FUNCTION_BLOCK FB_Tote_Subsystem
VAR_INPUT
END_VAR
VAR_OUTPUT
END_VAR
VAR
	status	: MachineStatus := MachineStatus.STOPPED;
	workflow_status	: ToteSubsystemWorkflowStatus := ToteSubsystemWorkflowStatus.UNKNOWN;
	error_status	: OrderToteErrorStatus := OrderToteErrorStatus.UNKNOWN;
	loading_tote	: FB_ToteData;
	buffer_tote		: FB_ToteData;
	working_tote	: FB_ToteData;
	machine_control_cmd	: MachineControlCommand;

	cmd	: OrderToteCommand;
	iLoad	: INT;
	iUnload	: INT;
	ton1	: TON;
	working_tote_status	: ToteStatus;
	p_eTransfer_working	: POINTER TO E_Transfer;

END_VAR


//status					:= GVL.machine_status;
workflow_status			:= GVL.fb_working.workflow_status;
error_status			:= GVL.fb_working.error_status;
working_tote._status	:= GVL.fb_working.tote_status;

p_eTransfer_working	:= ADR(GVL.fb_working.eTransfer);
CASE cmd OF
	OrderToteCommand.DO_NOTHING:
		p_eTransfer_working^	:= E_Transfer.IDLE;
	OrderToteCommand.LOAD:
		p_eTransfer_working^	:= E_Transfer.LOAD;
		IF GVL.fb_working.M_load() THEN
			cmd	:= OrderToteCommand.DO_NOTHING;
		END_IF
	OrderToteCommand.OPEN_BAG:
		workflow_status := ToteSubsystemWorkflowStatus.BAG_OPENING;
		working_tote._status	:= ToteStatus.READY;
		workflow_status := ToteSubsystemWorkflowStatus.IDLE;
		IF GVL.fb_working.M_bag_open() THEN
			cmd	:= OrderToteCommand.DO_NOTHING;
		END_IF
		
	;
	OrderToteCommand.STOP:
		working_tote._status	:= ToteStatus.EMPTY;
		workflow_status := ToteSubsystemWorkflowStatus.IDLE;
		cmd	:= OrderToteCommand.DO_NOTHING;
		;
	OrderToteCommand.SWAP:
		IF M_Unload() THEN
			IF M_Load() THEN
				cmd	:= OrderToteCommand.DO_NOTHING;
			END_IF
		END_IF
	;
	OrderToteCommand.UNLOAD:
		p_eTransfer_working^	:= E_Transfer.UNLOAD;
		IF GVL.fb_working.M_unload() THEN
			cmd	:= OrderToteCommand.DO_NOTHING;
		END_IF
	;	
END_CASE
ton1(PT:=T#1S);

METHOD M_Load : BOOL
VAR_INPUT
END_VAR
M_Load	:=FALSE;
CASE iLoad OF
	0:	
		working_tote._status	:= ToteStatus.EMPTY;
		workflow_status := ToteSubsystemWorkflowStatus.WAITING_FOR_NEW_TOTE;
		ton1.IN	:= FALSE;
		//GVL.iLoad	:= 1;
	1:
		ton1.IN	:= TRUE;
		IF ton1.Q THEN
			ton1.IN	:= FALSE;
			iLoad	:= 2;
		END_IF
	2:	
		workflow_status := ToteSubsystemWorkflowStatus.INBOUNDING;
		working_tote._status	:= ToteStatus.LOADED;
		iLoad	:= 3;
	3:
		ton1.IN	:= TRUE;
		IF ton1.Q THEN
			ton1.IN	:= FALSE;
			iLoad	:= 4;
		END_IF
	4:	
		workflow_status := ToteSubsystemWorkflowStatus.BAG_OPENING;
		working_tote._status	:= ToteStatus.READY;
		iLoad	:= 5;
	5:
		ton1.IN	:= TRUE;
		IF ton1.Q THEN
			ton1.IN	:= FALSE;
			iLoad	:= 6;
		END_IF		
	6:	
		workflow_status := ToteSubsystemWorkflowStatus.IDLE;
		iLoad	:= 0;
		M_Load	:= TRUE;
		GVL.fb_working.M_load();
END_CASE
END_METHOD

METHOD M_Swap : BOOL
VAR_INPUT
END_VAR
END_METHOD

METHOD M_Unload : BOOL
VAR_INPUT
END_VAR
M_Unload	:=FALSE;
CASE iUnload OF	
	0:	
		workflow_status := ToteSubsystemWorkflowStatus.WAITING_FOR_UNLOADING;
		ton1.IN	:= FALSE;
		iUnload	:= 1;
	1:
		ton1.IN	:= TRUE;
		IF ton1.Q THEN
			ton1.IN	:= FALSE;
			iUnload	:= 2;
		END_IF
	2:	
		workflow_status := ToteSubsystemWorkflowStatus.OUTBOUNDING;
		working_tote._status	:= ToteStatus.EMPTY;
		iUnload	:= 3;
	3:
		ton1.IN	:= TRUE;
		IF ton1.Q THEN
			ton1.IN	:= FALSE;
			iUnload	:= 4;
		END_IF	
	4:	
		workflow_status := ToteSubsystemWorkflowStatus.IDLE;
		iUnload	:= 0;
		M_Unload	:=TRUE;
END_CASE
END_METHOD

{attribute 'TcRpcEnable'}
METHOD machine_control_command : BOOL
VAR_INPUT
	Command	: MachineControlCommand;
END_VAR
machine_control_command	:= FALSE; 

machine_control_cmd	:= Command;

machine_control_command	:= TRUE;
END_METHOD

{attribute 'TcRpcEnable'}
METHOD order_tote_action_request : BOOL
VAR_INPUT
	Command	: OrderToteCommand;
END_VAR
order_tote_action_request	:= FALSE; 
IF MAIN.eState=E_SystemManager.IN_PROGRESS AND cmd=OrderToteCommand.DO_NOTHING THEN
	cmd	:= Command;
ELSE
	error_status	:= OrderToteErrorStatus.MACHINE_NOT_RUNNING;
	cmd	:= OrderToteCommand.DO_NOTHING;
END_IF

order_tote_action_request	:= TRUE;
END_METHOD

END_FUNCTION_BLOCK

(* stored: Version 1.1.0.1, ProductVersion 3.1.4024.12
   POU FB_Tote_Subsystem: Id {18f3e813-8d9e-4f02-997f-31b8e26895c7}, SpecialFunc None
   Method M_Load: Id {f3d31d0d-ba45-4048-bf50-b51644cf2466}
   Method M_Swap: Id {20428881-b3c0-40e9-9ad8-a4eb281ff8b2}
   Method M_Unload: Id {3b2ff3c1-e38e-4c29-abd4-860eb0b1090d}
   Method machine_control_command: Id {e35d6b29-fce8-4046-8fa5-9d1764fae381}
   Method order_tote_action_request: Id {070e3305-f432-4c7a-8094-5803fe668fc5} *)
